FUNCTION_BLOCK XtsMover
VAR
END_VAR

METHOD Disable : BOOL
VAR_INPUT
END_VAR
END_METHOD

METHOD Enable : BOOL
VAR_INPUT
END_VAR
END_METHOD

METHOD MoveTo : BOOL
VAR_INPUT
END_VAR
END_METHOD

METHOD Reset : BOOL
VAR_INPUT
END_VAR
END_METHOD

END_FUNCTION_BLOCK

(* stored: Version 1.1.0.1, ProductVersion 3.1.4024.12
   POU XtsMover: Id {1fb5bd84-a3b2-48b8-baa6-4a91754a9048}, SpecialFunc None
   Method Disable: Id {cf9f3eee-1dc6-4244-a951-8c14201d03a0}
   Method Enable: Id {7aed0b8f-bc77-4a99-a38a-4bc2ad677d35}
   Method MoveTo: Id {c35c82b9-4c37-4510-8280-f515e355ba6f}
   Method Reset: Id {3b6bb063-5916-411c-8ff0-b290db583cee} *)
